PROGRAM BASE64_DEMO_1
VAR
	text1: STRING(144) := '<4036.1076324381@guildenstern.zeitform.de>';
	text2: STRING(192);
	text3: STRING(144);
	BASE64_DECODE_STR: BASE64_DECODE_STR;
	BASE64_ENCODE_STR: BASE64_ENCODE_STR;
	start: BOOL := TRUE;
	done1: BOOL;
	done2: BOOL;
END_VAR

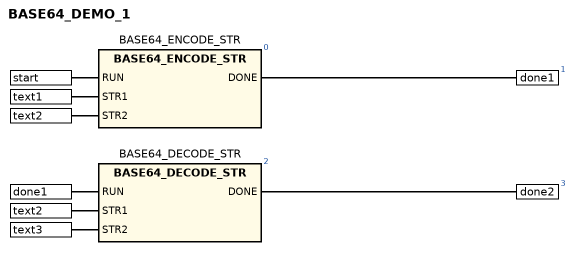
BASE64_ENCODE_STR(RUN := start, STR1 := text1, STR2 := text2);
done1 := BASE64_ENCODE_STR.DONE;
BASE64_DECODE_STR(RUN := done1, STR1 := text2, STR2 := text3);
done2 := BASE64_DECODE_STR.DONE;

END_PROGRAM

(* stored: Version 1.1.0.1, ProductVersion 3.1.4024.0
   POU BASE64_DEMO_1: Id {a5efec1e-a3ec-4ced-b5b4-efb44090b2a7}, SpecialFunc None *)
